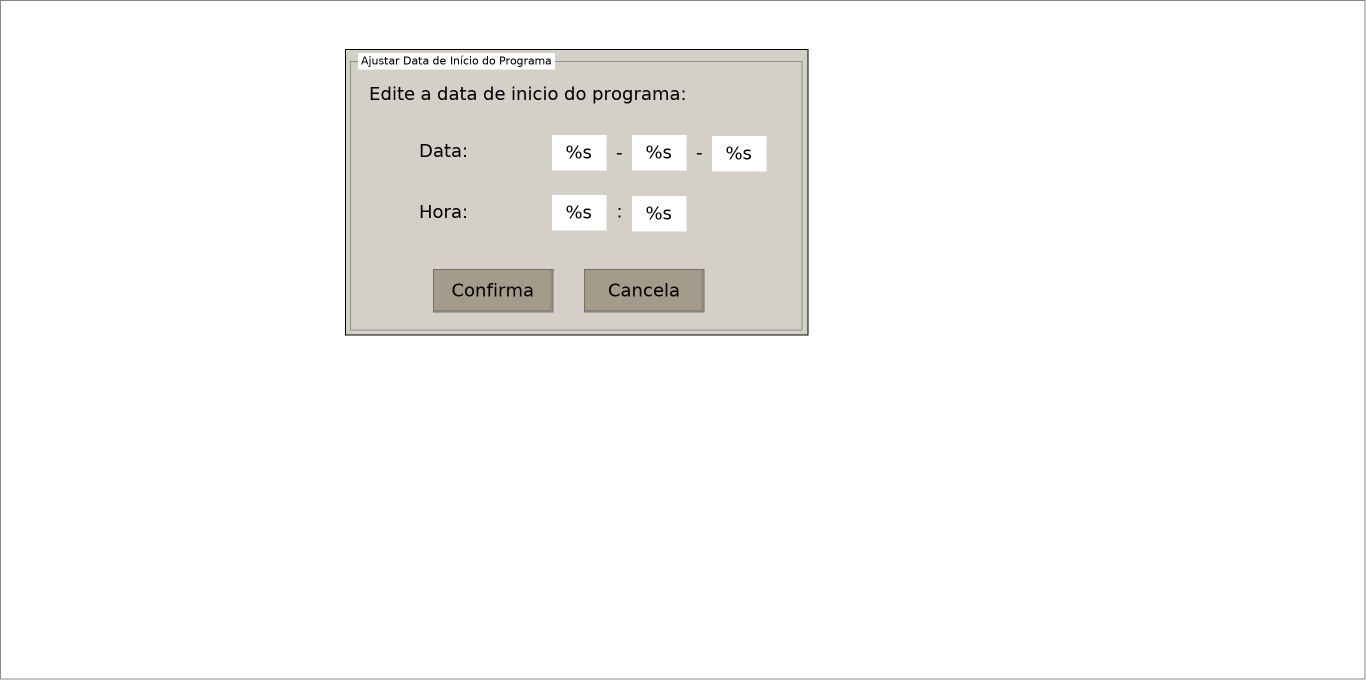
VISUALIZATION setInicio  // 1366x680
    Rectangle (345,49 463x286)
    GroupBox (350,53 452x277), "Ajustar Data de Início do Programa"
        Label (16,25 316x32), "Edite a data de inicio do programa:"
        Textfield (281,81 56x37), "%s", text variable: GVL.mes
            OnMouseClick: write the text variable via VisuDialogs.Numpad
        Textfield (361,82 56x37), "%s", text variable: GVL.ano
            OnMouseClick: write the text variable via VisuDialogs.Numpad
        Textfield (201,141 56x37), "%s", text variable: GVL.hora
            OnMouseClick: write the text variable via VisuDialogs.Numpad
        Textfield (281,142 56x37), "%s", text variable: GVL.minuto
            OnMouseClick: write the text variable via VisuDialogs.Numpad
        Label (35,144 86x30), "Hora:"
        Label (338,82 23x35), "-"
        Label (258,141 23x35), ":"
        Button (83,216 120x43), "Confirma"
            OnMouseClick: CloseDialog Dialog=setInicio, Result=OK, NumpadKeypadSet=True
            OnMouseClick: execute { confirmSetInicio(); }
        Button (234,216 120x43), "Cancela"
            OnMouseClick: CloseDialog Dialog=setInicio, Result=Cancel, NumpadKeypadSet=True
    Textfield (551,134 56x37), "%s", text variable: GVL.dia
        OnMouseClick: write the text variable via VisuDialogs.Numpad
    Label (385,136 86x30), "Data:"
    Label (608,135 23x35), "-"
END_VISUALIZATION
